(*
  FB_PompDrukPID
  ==============
  PI(D) regelaar voor pompdrukregeling in TwinCAT 3.

  Regelstrategie:
    - P : Proportioneel — directe reactie op afwijking
    - I : Integraal     — elimineert blijvende afwijking (steady-state error)
    - D : Differentieel — standaard UIT (Td = 0).
          D versterkt sensorruis en is voor pompdruk niet aanbevolen.

  Blip-vrij (bumpless transfer):
    Bij inschakelen en bij reset wordt het integraal voorgeladen zodat de
    uitgang vloeiend start op 0 zonder schok.

  Setpoint ramp:
    rSpRamp [bar/s] begrenst hoe snel het interne setpoint mag wijzigen.
    Voorkomt P-piek bij grote setpointsprongen. 0.0 = ramp uitgeschakeld.

  Hysterese op aan/uit schakeldrempel (anti-puls):
    Pomp gaat UIT als PID-uitgang < rUitMin.
    Pomp gaat AAN pas als PID-uitgang >= rUitMin + rHysterese.
    Voorkomt pulsen/klapperen bij overshoot terugkeer naar setpoint.
    Anti-windup respecteert de hysterese: integraal stopt ook tijdens
    de hysteresezone zodat de drempel niet herhaaldelijk geraakt wordt.

  Anti-windup:
    Integraal stopt met opladen wanneer de pomp gesatureerd is
    (uitgang = 0 of uitgang = rUitMax) in dezelfde richting als de afwijking.

  Parameters:
    bEnable       : PID actief. Bij FALSE: uitgang = 0, bumpless tracking.
    rSetpoint     : Gewenste druk [bar]
    rMeting       : Gemeten druk van sensor [bar]
    rKp           : Proportionele versterking [-]
    rTi           : Integratietijd [s]  — 0.0 = integraal uitgeschakeld
    rTd           : Differentiatietijd [s] — 0.0 = differentiaal uitgeschakeld (aanbevolen)
    rSpRamp       : Max setpointwijziging [bar/s] — 0.0 = ramp uitgeschakeld
    rUitMin       : Minimale pompuitgang als pomp loopt [%]
    rUitMax       : Maximale pompuitgang [%]
    rHysterese    : Hysterese boven rUitMin voor inschakelen [%] (aanbevolen: 3-10%)
    rCyclustijd   : PLC taskperiode [s]  (bv. 0.01 voor 10ms task)
    bReset        : Stijgende flank: bumpless reset naar 0
*)
FUNCTION_BLOCK FB_PompDrukPID
VAR_INPUT
    bEnable       : BOOL;                 // PID inschakelen
    rSetpoint     : REAL;                 // Gewenste druk [bar]
    rMeting       : REAL;                 // Gemeten druk [bar]
    rKp           : REAL := 5.0;          // Proportionele versterking [-]
    rTi           : REAL := 2.0;          // Integratietijd [s]  (0 = I uit)
    rTd           : REAL := 0.0;          // Differentiatietijd [s] (0 = D uit, aanbevolen)
    rSpRamp       : REAL := 0.0;          // Max setpointwijziging [bar/s] (0 = uit)
    rUitMin       : REAL := 0.0;          // Minimum pompuitgang als pomp loopt [%]
    rUitMax       : REAL := 100.0;        // Maximum pompuitgang [%]
    rHysterese    : REAL := 5.0;          // Hysterese boven rUitMin voor inschakelen [%]
    rCyclustijd   : REAL := 0.01;         // Taskperiode [s]
    bReset        : BOOL;                 // Bumpless reset naar 0
END_VAR
VAR_OUTPUT
    rUitgang        : REAL;               // Pompuitgang [%]  (0 of rUitMin..rUitMax)
    bPompLoopt      : BOOL;               // TRUE = pomp draait
    rSetpointActief : REAL;               // Intern (gerampte) setpoint [bar]
    rAfwijking      : REAL;               // Regelafwijking: setpoint - meting [bar]
    rPDeel          : REAL;               // P-bijdrage [%]
    rIDeel          : REAL;               // I-bijdrage [%]
    rDDeel          : REAL;               // D-bijdrage [%]
    bMaxBegrensd    : BOOL;               // Uitgang begrensd op maximum
END_VAR
VAR
    rIntegraal      : REAL;               // Integraalsom
    rMetingVorig    : REAL;               // Meting vorige cyclus (voor D op meting)
    rUitOngeclipped : REAL;               // PID som voor begrenzing
    bResetVorig     : BOOL;               // Flankdetectie reset
    rSpIntern       : REAL;               // Gerampte setpoint intern
    bEersteRun      : BOOL := TRUE;       // Initialisatie eerste scan
END_VAR


// --- Initialisatie eerste scan ---
IF bEersteRun THEN
    rSpIntern    := rSetpoint;
    rMetingVorig := rMeting;
    bEersteRun   := FALSE;
END_IF

// --- Veiligheidscontrole parameters ---
IF rCyclustijd <= 0.0 THEN rCyclustijd := 0.01; END_IF
IF rUitMax <= rUitMin  THEN rUitMax    := rUitMin + 1.0; END_IF
IF rHysterese < 0.0    THEN rHysterese := 0.0; END_IF

// --- Setpoint ramp (begrenst sprongen op setpoint) ---
IF rSpRamp > 0.0 THEN
    IF rSetpoint > rSpIntern + rSpRamp * rCyclustijd THEN
        rSpIntern := rSpIntern + rSpRamp * rCyclustijd;
    ELSIF rSetpoint < rSpIntern - rSpRamp * rCyclustijd THEN
        rSpIntern := rSpIntern - rSpRamp * rCyclustijd;
    ELSE
        rSpIntern := rSetpoint;
    END_IF
ELSE
    rSpIntern := rSetpoint;
END_IF
rSetpointActief := rSpIntern;

// --- Regelafwijking (ook berekend als PID uit, voor bumpless tracking) ---
rAfwijking := rSpIntern - rMeting;
rPDeel     := rKp * rAfwijking;

// --- Bumpless reset op stijgende flank ---
IF bReset AND NOT bResetVorig THEN
    IF rTi > 0.0 AND rKp > 0.0 THEN
        rIntegraal := (0.0 - rPDeel) * rTi / rKp;
    ELSE
        rIntegraal := 0.0;
    END_IF
    rMetingVorig := rMeting;
    bPompLoopt   := FALSE;
END_IF
bResetVorig := bReset;

// --- PID inactief: uitgang = 0, integraal tracken voor bumpless inschakelen ---
IF NOT bEnable THEN
    rSpIntern       := rSetpoint;
    rSetpointActief := rSpIntern;

    IF rTi > 0.0 AND rKp > 0.0 THEN
        rIntegraal := (0.0 - rPDeel) * rTi / rKp;
    ELSE
        rIntegraal := 0.0;
    END_IF
    rMetingVorig := rMeting;
    bPompLoopt   := FALSE;

    rUitgang     := 0.0;
    rIDeel       := 0.0;
    rDDeel       := 0.0;
    bMaxBegrensd := FALSE;
    RETURN;
END_IF

// --- I-deel met anti-windup ---
// bPompLoopt=FALSE betekent uitgang=0 (pomp uit of in hysteresezone)
// Stop negatief integreren als pomp uit is, stop positief als max bereikt
IF rTi > 0.0 THEN
    IF NOT (bMaxBegrensd   AND rAfwijking > 0.0)
    AND NOT (NOT bPompLoopt AND rAfwijking < 0.0) THEN
        rIntegraal := rIntegraal + rAfwijking * rCyclustijd;
    END_IF
    rIDeel := (rKp / rTi) * rIntegraal;
ELSE
    rIntegraal := 0.0;
    rIDeel     := 0.0;
END_IF

// --- D-deel op meting (vermijdt D-kick bij setpointwijziging) ---
IF rTd > 0.0 THEN
    rDDeel := -rKp * rTd * (rMeting - rMetingVorig) / rCyclustijd;
ELSE
    rDDeel := 0.0;
END_IF
rMetingVorig := rMeting;

// --- PID som ---
rUitOngeclipped := rPDeel + rIDeel + rDDeel;

// --- Uitgang met hysterese op inschakelpunt ---
//
//   Pomp UIT  -> AAN : uitgang moet >= rUitMin + rHysterese bereiken
//   Pomp AAN  -> UIT : uitgang daalt onder rUitMin
//
//   Zo wordt klapperen/pulsen tijdens overshoot-terugkeer voorkomen:
//   de pomp start pas opnieuw als de PID duidelijk boven de drempel zit.
//
bMaxBegrensd := rUitOngeclipped > rUitMax;

IF rUitOngeclipped < rUitMin THEN
    // Uitgang onder minimum: pomp volledig uit
    rUitgang   := 0.0;
    bPompLoopt := FALSE;

ELSIF NOT bPompLoopt AND rUitOngeclipped < rUitMin + rHysterese THEN
    // Pomp was uit en uitgang zit in de hysteresezone: nog niet inschakelen
    rUitgang   := 0.0;
    bPompLoopt := FALSE;

ELSIF bMaxBegrensd THEN
    // Uitgang boven maximum: begrensd
    rUitgang   := rUitMax;
    bPompLoopt := TRUE;

ELSE
    // Normaal bedrijf: rUitMin <= uitgang <= rUitMax
    rUitgang   := rUitOngeclipped;
    bPompLoopt := TRUE;
END_IF

END_FUNCTION_BLOCK

(* stored: Version 1.1.0.1, ProductVersion 3.1.4024.0
   POU FB_PompDrukPID: Id {a1b2c3d4-e5f6-7890-abcd-ef1234567890}, SpecialFunc None *)
